{attribute 'TcGenerated'}
{attribute 'no-analysis'}
{attribute 'linkalways'}
// This function has been automatically generated from the project information.
VAR_GLOBAL CONSTANT
	{attribute 'const_non_replaced'}
	stLibVersion_CNM_AssertionInterfaceTests : ST_LibVersion := (iMajor := 1, iMinor := 0, iBuild := 0, iRevision := 47, nFlags := 0, sVersion := '1.0.0.47');
END_VAR

(* stored: Version 1.1.0.1, ProductVersion 3.1.4024.12
   GVL Global_Version: Id {91371787-d2b0-4009-99b2-9d1d271cb382} *)
